INTERFACE I_CalcFocalLengthSingleLens EXTENDS I_Fallible


METHOD Calculate : LREAL
VAR_INPUT
    sElementName : STRING;
    fRadius : LREAL;
END_VAR
END_METHOD

END_INTERFACE

(* stored: Version 1.1.0.1
   Itf I_CalcFocalLengthSingleLens: Id {e12f78e2-8770-4788-8553-7f4967f11469}
   Method Calculate: Id {dd290774-7390-4466-a975-f33897623e2d} *)
